FUNCTION_BLOCK ConveyorCTL_Multicast (* Basic Function Block Type *)
  (* Standard: 61499-2 *)
  (* Version 0.2, 2003-12-04, JHC, Rockwell Automation, Renamed for better indexing. *)
  (* Version 0.1, 2002-11-05, JHC, Rockwell Automation, Corrected missing ST element in Algorithm REQ. *)
  (* Version 0.0, 2000-05-30, JHC, Rockwell Automation *)
  (* Compiler header: package fb.rt.cs725; *)
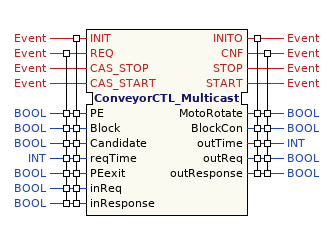
  EVENT_INPUT
    INIT WITH PE, Block, Candidate, reqTime, PEexit, inReq, inResponse; (* Initialization Request *)
    REQ WITH PE, Block, Candidate, reqTime, PEexit, inReq, inResponse; (* Normal Execution Request *)
    CAS_STOP;
    CAS_START;
  END_EVENT
  EVENT_OUTPUT
    INITO WITH MotoRotate, BlockCon, outTime, outReq, outResponse; (* Initialization Confirm *)
    CNF WITH MotoRotate, BlockCon, outTime, outReq, outResponse; (* Execution Confirmation *)
    STOP;
    START;
  END_EVENT
  VAR_INPUT
    PE : BOOL; (* Input event qualifier *)
    Block : BOOL;
    Candidate : BOOL;
    reqTime : INT;
    PEexit : BOOL;
    inReq : BOOL;
    inResponse : BOOL;
  END_VAR
  VAR_OUTPUT
    MotoRotate : BOOL; (* Output event qualifier *)
    BlockCon : BOOL;
    outTime : INT;
    outReq : BOOL;
    outResponse : BOOL;
  END_VAR
  VAR
    lastPE : BOOL := 1;
    lastBlock : BOOL := 0;
    state : INT := 0;
    timeStamp : INT := 0;
    savedReqTime : INT := 0;
    waitFlag : BOOL := false;
  END_VAR
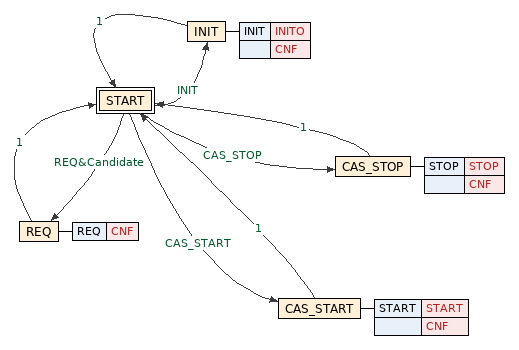
  EC_STATES
    START; (* Initial State *)
    INIT : INIT -> INITO, -> CNF; (* Initialization *)
    REQ : REQ -> CNF; (* Normal execution *)
    CAS_START : START -> START, -> CNF;
    CAS_STOP : STOP -> STOP, -> CNF;
  END_STATES
  EC_TRANSITIONS
    START TO INIT := INIT;
    INIT TO START := 1;
    START TO REQ := REQ&Candidate;
    REQ TO START := 1;
    START TO CAS_START := CAS_START;
    CAS_START TO START := 1;
    START TO CAS_STOP := CAS_STOP;
    CAS_STOP TO START := 1;
  END_TRANSITIONS
  ALGORITHM INIT IN Java: (* Initialization algorithm *)
MotoRotate.value=true;
Block.value=false;
outTime.value =0;
outReq.value =false;
outResponse.value =false;

System.out.println(this+" "+MotoRotate.value);
System.out.println(MotoRotate.value);
  END_ALGORITHM
  ALGORITHM REQ IN Java: (* Normally executed algorithm *)
//state = 0,1,2 (released,wanted,held)

if (Candidate.value) {
 if (inResponse.value) {
     waitFlag.value = true;
  state.value = 2;
 } else if (!PE.value) {
  state.value = 1;
 } else {
     waitFlag.value = true;
  state.value = 0;
 }

  if (lastBlock.value != Block.value) {
   if (Block.value) {
    STOP.serviceEvent(this);
    MotoRotate.value = false;
    System.out.println("Cas Stop");
   } else {
    START.serviceEvent(this);
    MotoRotate.value = true;
    System.out.println("Cas Start");

   }
   lastBlock.value = Block.value;
  }

 if (state.value == 0) {
  outReq.value = false;
  BlockCon.value = false;
  MotoRotate.value = true;
  if (inReq.value) {
   outResponse.value = true;
  }
  else {
      outResponse.value = false;
  }
    System.out.println("CONVEYOR IS IN THE RELEASED STATE-----------------------------");

 }
 else if (state.value == 1) {
     if (waitFlag.value) {
          savedReqTime.value = timeStamp.value;
          waitFlag.value = false;
     }
System.out.println("SAVED TIME IS --------------------- " + savedReqTime);

  outReq.value = true;
  outTime.value = timeStamp.value;
  BlockCon.value = true;
  MotoRotate.value = false;
  if (inReq.value) {
   if (reqTime.value < savedReqTime.value) {
    outResponse.value = true;
    BlockCon.value = true;
    MotoRotate.value = false;

   } else {
    outResponse.value = false;
    outReq.value = false;
    BlockCon.value = false;
    MotoRotate.value = true;
    state.value = 2;
        System.out.println("CONVEYOR IS IN THE WAITING STATE-----------------------------");

   }
  }

    System.out.println("CONVEYOR IS IN THE WAITING STATE-----------------------------");

 }
 else {
  outReq.value = false;
  BlockCon.value = false;
  outResponse.value = false;

  if (!PEexit.value && PE.value) {
      state.value = 0;
  }
  else if (!PEexit.value && !PE.value) {
      state.value = 1;
  }

  System.out.println("CONVEYOR IS IN THE HELD STATE-----------------------------");
 }
}

timeStamp.value++;
  END_ALGORITHM
  ALGORITHM START IN ST:
MotoRotate:=TRUE;
System.out.println(this + "//////////////////////////////////////////////////////////////// Start " + MotoRotate);
  END_ALGORITHM
  ALGORITHM STOP IN ST:
MotoRotate := FALSE;
System.out.println(this + "/////////////////////////////////////////////////// Stop " + MotoRotate);
  END_ALGORITHM
END_FUNCTION_BLOCK
